FUNCTION ifExprFunc2: BOOL
VAR_INPUT
    farg_f2_p: BOOL;
END_VAR


        IF (farg_f2_p) THEN
    ifExprFunc2 := TRUE;
ELSE
    ifExprFunc2 := TRUE;
END_IF;

END_FUNCTION

(* stored: ProductVersion 3.1.0.18, Version 1.1.0.1 *)
